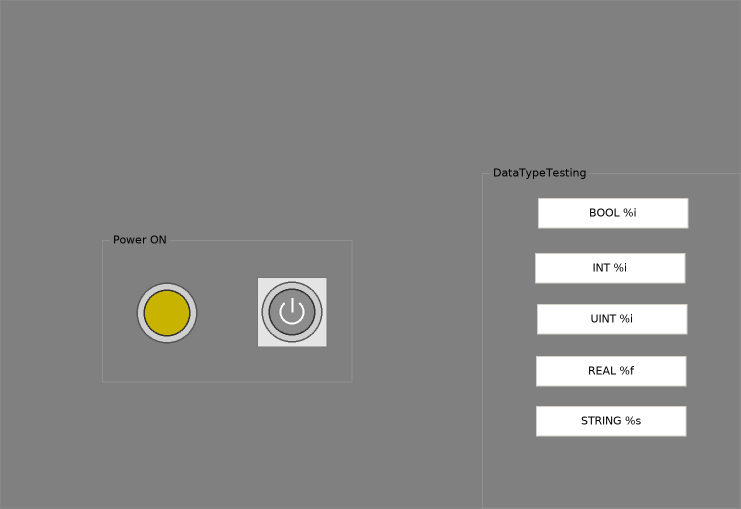
VISUALIZATION HMI  // 741x509
    GroupBox (102,232 250x150), "Power ON"
        Lamp1 (30,46 70x70), variable: MAIN.bEnable, style: Lamp-Lamp1-Yellow
        PowerSwitch (155,45 70x70), variable: MAIN.bStart, behaviour: TOGGLE, style: Switch-PowerSwitch-Gray
    GroupBox (482,165 259x344), "DataTypeTesting"
        Textfield (56,33 150x30), "BOOL %i", text variable: MAIN.bEnable
        Textfield (53,88 150x30), "INT %i", text variable: MAIN.nINT
        Textfield (55,139 150x30), "UINT %i", text variable: MAIN.nUINT
        Textfield (54,191 150x30), "REAL %f", text variable: MAIN.fREAL
        Textfield (54,241 150x30), "STRING %s", text variable: MAIN.sPowerStatus
            OnMouseDown: write the text variable via Default
END_VISUALIZATION

(* stored: Version 1.1.0.1, ProductVersion 3.1.4024.12
   Visu HMI: Id {e9ee8fbe-e49f-4f21-b26d-b9808343ec41} *)
